FUNCTION_BLOCK FB_DataChannelSenderFifo EXTENDS FB_DynamicFifo
VAR
	m_pDataChannel: POINTER TO FB_DataChannelSendBase;
	m_pItem: POINTER TO BYTE;
	m_bolEnable: BOOL;
	m_intMaxFifoSize: INT := 10;
	bResult: BOOL;
END_VAR

IF (m_uinItemCount > 0) AND NOT m_pDataChannel^.Busy THEN
	m_pItem := Pop();

	IF m_bolEnable THEN
		bResult := m_pDataChannel^.SendData(
						pData       := m_pItem,
						udiDataSize := m_pDataChannel^.DataSize);
	END_IF;
	
	IF m_bFreeDataPointer THEN
		__DELETE(m_pItem);
	END_IF
END_IF

IF m_pDataChannel^.ClearBufferRequest THEN
	THIS^.ClearFifo();
	m_pDataChannel^.ClearBufferDone();
END_IF

m_pDataChannel^();

PROPERTY Enable : BOOL
SET
IF m_bolEnable AND NOT Enable THEN
	THIS^.ClearFifo();
END_IF

m_bolEnable := Enable;
END_SET
GET
Enable := m_bolEnable;
END_GET
END_PROPERTY

PROPERTY MaxFifoSize : INT
SET
m_intMaxFifoSize := MaxFifoSize;
END_SET
GET
MaxFifoSize := m_intMaxFifoSize;
END_GET
END_PROPERTY

PROPERTY DataChannel : POINTER TO FB_DataChannelSendBase
SET
m_pDataChannel := DataChannel;
END_SET
END_PROPERTY

END_FUNCTION_BLOCK

(* stored: Version 1.1.0.1, ProductVersion 3.1.0.26
   POU FB_DataChannelSenderFifo: Id {95a8c786-ddff-4f2b-8fcc-9ba2279e88fc}
   Property Enable: Id {6814a05e-0915-4ce7-9654-aa13af9283d8}
   Set Set: Id {0c066d85-60f0-4a32-878e-eef79f68c85b}
   Get Get: Id {0cf38208-7b99-4217-a5ef-daaf1f0ad964}
   Property MaxFifoSize: Id {83f7dfc5-778d-4cb9-a6dc-0069b04106d8}
   Set Set: Id {6770f965-a959-4db9-a564-af3808118cf9}
   Get Get: Id {af3b8be9-4a39-4a29-bd20-c561176dceba}
   Property DataChannel: Id {c6222d3b-7199-4e49-aac3-c195e3c27652}
   Set Set: Id {cc0198b0-85e5-4cba-a57f-b2ac53ff8f44} *)
